FUNCTION_BLOCK FB_Blinker_RD
VAR_INPUT
	OnTime							: TIME;					//On时长
	OffTime				   		: TIME;					//Off时长
END_VAR

VAR_OUTPUT
	clock							: BOOL;					//
	R_Plus						: BOOL;					//脉冲上升沿
	F_Plus						: BOOL;					//脉冲下降沿
END_VAR

VAR
	{attribute 'hide'}
	tonOff						: TON;					//Off计时器
	{attribute 'hide'}
	tonOn						: TON;					//On计时器
END_VAR

tonOff(IN:=NOT clock, PT:=OffTime, Q=>R_Plus );
tonOn(IN:=clock, PT:=OnTime, Q=>F_Plus );

IF R_Plus OR F_Plus THEN
	clock:= NOT clock;
END_IF

END_FUNCTION_BLOCK

(* stored: Version 1.1.0.1, ProductVersion 3.1.4024.12
   POU FB_Blinker_RD: Id {af2dfb15-ef1c-4ed4-acf7-63a146640b48}, SpecialFunc None *)
